INTERFACE I_FallibleINT EXTENDS I_Fallible

PROPERTY Val : INT
GET
END_GET
SET
END_SET
END_PROPERTY

END_INTERFACE

(* stored: Version 1.1.0.1, ProductVersion 3.1.4022.18
   Itf I_FallibleINT: Id {9aed38e0-684d-430f-a26a-a236f4e39527}
   Property Val: Id {86952b0e-9d30-4a56-89f3-07afe624326d}
   Get Get: Id {ccc13ada-480b-4804-9ff5-c11adbb234ef}
   Set Set: Id {f522d0d5-c1d5-440d-a23e-58e1d8e39a7d} *)
